PROGRAM StringsAndStructs

END_PROGRAM

(* stored: Version 1.1.0.1
   POU StringsAndStructs: Id {8d8e914b-dbd1-4e69-8633-8e0d76e9ab04}, SpecialFunc None *)
